// TIA Portal V19 export
ORGANIZATION_BLOCK "Main"   // OB1, LAD, ProgramCycle
TITLE = "Main Program Sweep (Cycle)"
{ S7_Optimized_Access := 'TRUE' }
// stored: SetENOAutomatically false
   VAR_INPUT
      Initial_Call : Bool;   // Initial call of this OB
      Remanence : Bool;   // =True, if remanent data are available
   END_VAR
   VAR_TEMP   // added for the SCL form of the ladder/FBD networks
      _w1 : Bool;
      _w2 : Bool;
   END_VAR
BEGIN

REGION Network 1
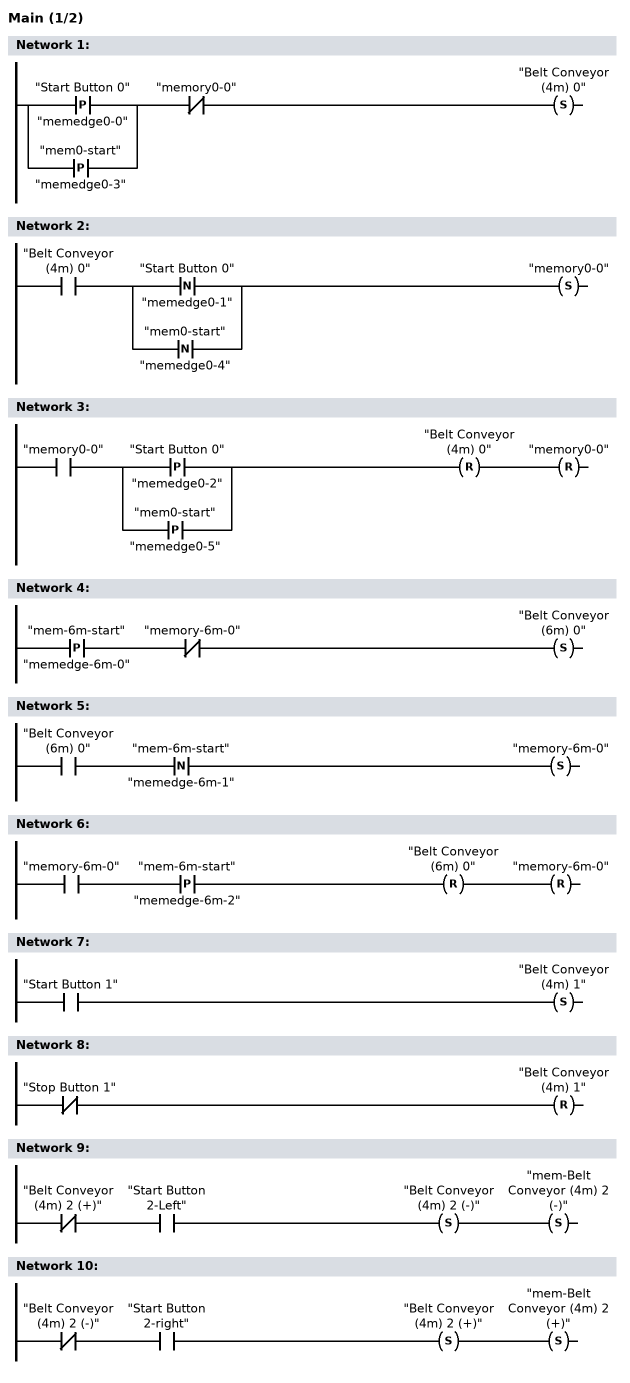
   RUNG wire#powerrail
      P_Contact(operand := "Start Button 0", bit := "memedge0-0")
      wire#w1
      I_Contact( "memory0-0" )
      S_Coil( "Belt Conveyor (4m) 0" )
   END_RUNG
   RUNG wire#powerrail
      P_Contact(operand := "mem0-start", bit := "memedge0-3")
   END_RUNG wire#w1
   // the same network as SCL:
   #_w1 := "Start Button 0" AND NOT "memedge0-0";   // rising edge of "Start Button 0"
   "memedge0-0" := "Start Button 0";
   #_w2 := "mem0-start" AND NOT "memedge0-3";   // rising edge of "mem0-start"
   "memedge0-3" := "mem0-start";
   IF (#_w1 OR #_w2) AND NOT "memory0-0" THEN "Belt Conveyor (4m) 0" := TRUE; END_IF;
END_REGION

REGION Network 2
   RUNG wire#powerrail
      Contact( "Belt Conveyor (4m) 0" )
      wire#w1
      N_Contact(operand := "Start Button 0", bit := "memedge0-1")
      wire#w2
      S_Coil( "memory0-0" )
   END_RUNG
   RUNG wire#w1
      N_Contact(operand := "mem0-start", bit := "memedge0-4")
   END_RUNG wire#w2
   // the same network as SCL:
   #_w1 := "Belt Conveyor (4m) 0" AND NOT "Start Button 0" AND "memedge0-1";   // falling edge of "Start Button 0"
   "memedge0-1" := "Start Button 0";
   #_w2 := "Belt Conveyor (4m) 0" AND NOT "mem0-start" AND "memedge0-4";   // falling edge of "mem0-start"
   "memedge0-4" := "mem0-start";
   IF #_w1 OR #_w2 THEN "memory0-0" := TRUE; END_IF;
END_REGION

REGION Network 3
   RUNG wire#powerrail
      Contact( "memory0-0" )
      wire#w1
      P_Contact(operand := "Start Button 0", bit := "memedge0-2")
      wire#w2
      R_Coil( "Belt Conveyor (4m) 0" )
      R_Coil( "memory0-0" )
   END_RUNG
   RUNG wire#w1
      P_Contact(operand := "mem0-start", bit := "memedge0-5")
   END_RUNG wire#w2
   // the same network as SCL:
   #_w1 := "memory0-0" AND "Start Button 0" AND NOT "memedge0-2";   // rising edge of "Start Button 0"
   "memedge0-2" := "Start Button 0";
   #_w2 := "memory0-0" AND "mem0-start" AND NOT "memedge0-5";   // rising edge of "mem0-start"
   "memedge0-5" := "mem0-start";
   IF #_w1 OR #_w2 THEN
       "Belt Conveyor (4m) 0" := FALSE;
       "memory0-0" := FALSE;
   END_IF;
END_REGION

REGION Network 4
   RUNG wire#powerrail
      P_Contact(operand := "mem-6m-start", bit := "memedge-6m-0")
      I_Contact( "memory-6m-0" )
      S_Coil( "Belt Conveyor (6m) 0" )
   END_RUNG
   // the same network as SCL:
   #_w1 := "mem-6m-start" AND NOT "memedge-6m-0";   // rising edge of "mem-6m-start"
   "memedge-6m-0" := "mem-6m-start";
   IF #_w1 AND NOT "memory-6m-0" THEN "Belt Conveyor (6m) 0" := TRUE; END_IF;
END_REGION

REGION Network 5
   RUNG wire#powerrail
      Contact( "Belt Conveyor (6m) 0" )
      N_Contact(operand := "mem-6m-start", bit := "memedge-6m-1")
      S_Coil( "memory-6m-0" )
   END_RUNG
   // the same network as SCL:
   #_w1 := "Belt Conveyor (6m) 0" AND NOT "mem-6m-start" AND "memedge-6m-1";   // falling edge of "mem-6m-start"
   "memedge-6m-1" := "mem-6m-start";
   IF #_w1 THEN "memory-6m-0" := TRUE; END_IF;
END_REGION

REGION Network 6
   RUNG wire#powerrail
      Contact( "memory-6m-0" )
      P_Contact(operand := "mem-6m-start", bit := "memedge-6m-2")
      R_Coil( "Belt Conveyor (6m) 0" )
      R_Coil( "memory-6m-0" )
   END_RUNG
   // the same network as SCL:
   #_w1 := "memory-6m-0" AND "mem-6m-start" AND NOT "memedge-6m-2";   // rising edge of "mem-6m-start"
   "memedge-6m-2" := "mem-6m-start";
   IF #_w1 THEN
       "Belt Conveyor (6m) 0" := FALSE;
       "memory-6m-0" := FALSE;
   END_IF;
END_REGION

REGION Network 7
   RUNG wire#powerrail
      Contact( "Start Button 1" )
      S_Coil( "Belt Conveyor (4m) 1" )
   END_RUNG
   // the same network as SCL:
   IF "Start Button 1" THEN "Belt Conveyor (4m) 1" := TRUE; END_IF;
END_REGION

REGION Network 8
   RUNG wire#powerrail
      I_Contact( "Stop Button 1" )
      R_Coil( "Belt Conveyor (4m) 1" )
   END_RUNG
   // the same network as SCL:
   IF NOT "Stop Button 1" THEN "Belt Conveyor (4m) 1" := FALSE; END_IF;
END_REGION

REGION Network 9
   RUNG wire#powerrail
      I_Contact( "Belt Conveyor (4m) 2 (+)" )
      Contact( "Start Button 2-Left" )
      S_Coil( "Belt Conveyor (4m) 2 (-)" )
      S_Coil( "mem-Belt Conveyor (4m) 2 (-)" )
   END_RUNG
   // the same network as SCL:
   IF NOT "Belt Conveyor (4m) 2 (+)" AND "Start Button 2-Left" THEN
       "Belt Conveyor (4m) 2 (-)" := TRUE;
       "mem-Belt Conveyor (4m) 2 (-)" := TRUE;
   END_IF;
END_REGION

REGION Network 10
   RUNG wire#powerrail
      I_Contact( "Belt Conveyor (4m) 2 (-)" )
      Contact( "Start Button 2-right" )
      S_Coil( "Belt Conveyor (4m) 2 (+)" )
      S_Coil( "mem-Belt Conveyor (4m) 2 (+)" )
   END_RUNG
   // the same network as SCL:
   IF NOT "Belt Conveyor (4m) 2 (-)" AND "Start Button 2-right" THEN
       "Belt Conveyor (4m) 2 (+)" := TRUE;
       "mem-Belt Conveyor (4m) 2 (+)" := TRUE;
   END_IF;
END_REGION

REGION Network 11
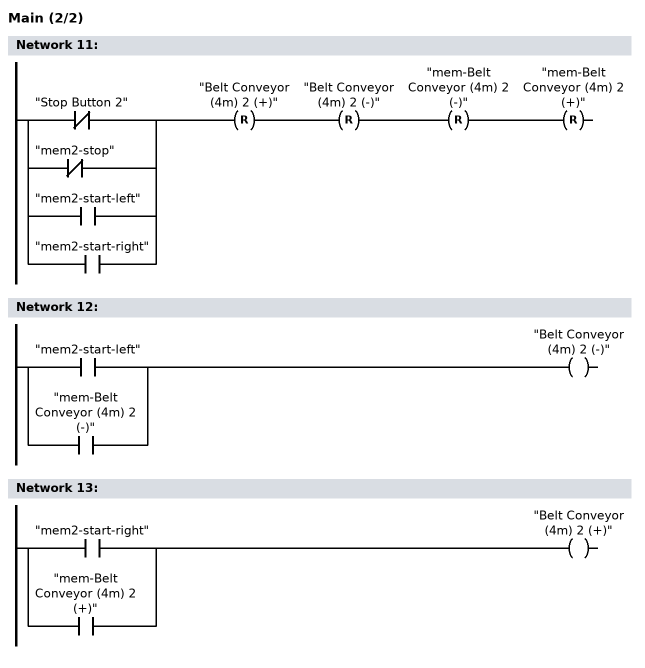
   RUNG wire#powerrail
      I_Contact( "Stop Button 2" )
      wire#w1
      R_Coil( "Belt Conveyor (4m) 2 (+)" )
      R_Coil( "Belt Conveyor (4m) 2 (-)" )
      R_Coil( "mem-Belt Conveyor (4m) 2 (-)" )
      R_Coil( "mem-Belt Conveyor (4m) 2 (+)" )
   END_RUNG
   RUNG wire#powerrail
      I_Contact( "mem2-stop" )
   END_RUNG wire#w1
   RUNG wire#powerrail
      Contact( "mem2-start-left" )
   END_RUNG wire#w1
   RUNG wire#powerrail
      Contact( "mem2-start-right" )
   END_RUNG wire#w1
   // the same network as SCL:
   IF NOT "Stop Button 2" OR NOT "mem2-stop" OR "mem2-start-left" OR "mem2-start-right" THEN
       "Belt Conveyor (4m) 2 (+)" := FALSE;
       "Belt Conveyor (4m) 2 (-)" := FALSE;
       "mem-Belt Conveyor (4m) 2 (-)" := FALSE;
       "mem-Belt Conveyor (4m) 2 (+)" := FALSE;
   END_IF;
END_REGION

REGION Network 12
   RUNG wire#powerrail
      Contact( "mem2-start-left" )
      wire#w1
      Coil( "Belt Conveyor (4m) 2 (-)" )
   END_RUNG
   RUNG wire#powerrail
      Contact( "mem-Belt Conveyor (4m) 2 (-)" )
   END_RUNG wire#w1
   // the same network as SCL:
   "Belt Conveyor (4m) 2 (-)" := "mem2-start-left" OR "mem-Belt Conveyor (4m) 2 (-)";
END_REGION

REGION Network 13
   RUNG wire#powerrail
      Contact( "mem2-start-right" )
      wire#w1
      Coil( "Belt Conveyor (4m) 2 (+)" )
   END_RUNG
   RUNG wire#powerrail
      Contact( "mem-Belt Conveyor (4m) 2 (+)" )
   END_RUNG wire#w1
   // the same network as SCL:
   "Belt Conveyor (4m) 2 (+)" := "mem2-start-right" OR "mem-Belt Conveyor (4m) 2 (+)";
END_REGION
END_ORGANIZATION_BLOCK
